# EPICS substitutions: powerlink/powerlinkApp/Db/userHost.substitutions
# Example substitutions file

file "db/dbExample1.db" {
    { user = "oplk-devHost" }
}

file db/dbExample2.db {
    pattern { user, no, scan }
        { "oplk-devHost", 1, "1 second" }
        { "oplk-devHost", 2, "2 second" }
        { "oplk-devHost", 3, "5 second" }
}
